TYPE ST_System_LA_Zustand :
STRUCT


	Betrieb_Anford			: BOOL;
	Betrieb_Soll				: BOOL;
	Betrieb					: BOOL;

	Modus_Heizung			: BOOL;
	Modus_Kuehlung			: BOOL;

	Netze_Anford				: ST_Zustand_Netze_Anford;

	Freigabe					: BOOL;
	Freigabe_Deakt			: BOOL;
	Freigabe_Code			: WORD;

	Stoerung					: BOOL;
	Stoerung_Code			: WORD;

	Warnung					: BOOL;
	Warnung_Code			: WORD;

	Status					: SINT;
	Status_Vorl_Pumpe		: BOOL;
	Status_Vorl_Regelventil	: BOOL;
	Status_Nachl_Pumpe		: BOOL;
	Status_Nachl_Regelventil	: BOOL;

	Quittierung				: BOOL;




END_STRUCT
END_TYPE

(* stored: Version 1.1.0.1, ProductVersion 3.1.4024.9
   DUT ST_System_LA_Zustand: Id {49abc9d0-af3b-47f6-8e53-40cb70706e43} *)
